(* PLC project Unnamed, Unknown Unnamed 1 *)
(* stored: creationDateTime 2021-12-21T18:23:51, modificationDateTime 2021-12-22T22:57:15 *)

TYPE datatype0 : ARRAY[1..10] OF BYTE;
END_TYPE

FUNCTION_BLOCK bot_detect
  VAR_INPUT
    IN : BOOL;
  END_VAR
  VAR
    BDGENR : UINT;
    M : BOOL;
    INIT : BOOL;
  END_VAR
  VAR_OUTPUT
    OUT : UDINT;
  END_VAR

            (* Initialize our random generator *)
(* This IF is called only the first time this *)
(* block executes *)
IF INIT = 0 THEN
  {time_t t;
  srand((unsigned) time(&t))}
  INIT := 1;
END_IF;

IF M = 0 and IN = 1 THEN
  (* Using pragma to write code directly in C. *)
  (* You can access your PLC program variables using *)
  (* GetFbVar(var,...) and SetFbVar(var,val,...) calls *)
  {SetFbVar(BDGENR,rand())}
  IF BDGENR > 4000 THEN
    {SetFbVar(OUT,1)}
  END_IF;
  IF BDGENR <= 4000 THEN
    {SetFbVar(OUT,0)}
  END_IF;
END_IF;
M := IN;
          
END_FUNCTION_BLOCK

FUNCTION_BLOCK bot_size_rand_generator
  VAR_INPUT
    IN : BOOL;
  END_VAR
  VAR
    BSZGENR : UINT;
    M : BOOL;
    INIT : BOOL;
  END_VAR
  VAR_OUTPUT
    OUT : UDINT;
  END_VAR

            (* Initialize our random generator *)
(* This IF is called only the first time this *)
(* block executes *)
IF INIT = 0 THEN
  {time_t t;
  srand((unsigned) time(&t))}
  INIT := 1;
END_IF;

IF M = 0 and IN = 1 THEN
  (* Using pragma to write code directly in C. *)
  (* You can access your PLC program variables using *)
  (* GetFbVar(var,...) and SetFbVar(var,val,...) calls *)
  {SetFbVar(BSZGENR,rand())}
  IF BSZGENR > 9000 THEN
    {SetFbVar(OUT,1)}
  END_IF;
  IF BSZGENR <= 9000 THEN
    {SetFbVar(OUT,0)}
  END_IF;
END_IF;
M := IN;
          
END_FUNCTION_BLOCK

FUNCTION_BLOCK bot_state_rand_generator
  VAR_INPUT
    IN : BOOL;
  END_VAR
  VAR
    BSGENR : UINT;
    M : BOOL;
    INIT : BOOL;
  END_VAR
  VAR_OUTPUT
    OUT : UDINT;
  END_VAR

            (* Initialize our random generator *)
(* This IF is called only the first time this *)
(* block executes *)
IF INIT = 0 THEN
  {time_t t;
  srand((unsigned) time(&t))}
  INIT := 1;
END_IF;

IF M = 0 and IN = 1 THEN
  (* Using pragma to write code directly in C. *)
  (* You can access your PLC program variables using *)
  (* GetFbVar(var,...) and SetFbVar(var,val,...) calls *)
  {SetFbVar(BSGENR,rand())}
  IF BSGENR > 4000 THEN
    {SetFbVar(OUT,1)}
  END_IF;
  IF BSGENR <= 4000 THEN
    {SetFbVar(OUT,0)}
  END_IF;
END_IF;
M := IN;
          
END_FUNCTION_BLOCK

PROGRAM BottleRefill
  VAR
    Start AT %IX0.0 : BOOL;
    Stop AT %IX0.1 : BOOL;
    System_On AT %QX0.0 : BOOL;
  END_VAR
  VAR
    TON0 : TON;
    Time_On1 : TIME;
    Time_On2 : TIME;
    Bot_Detect_State : BOOL;
    bot_size_rand_generator0 : bot_size_rand_generator;
    bot_state_rand_generator0 : bot_state_rand_generator;
    Bot_Size1 : BOOL;
    Bot_Size2 : BOOL;
    Bot_Size3 : BOOL;
    Bot_Size4 : BOOL;
    Bot_Size5 : BOOL;
    first_bot_state_bit : BYTE;
    second_bot_state_bit : BYTE;
    third_bot_state_bit : BYTE;
    fourth_bot_state_bit : BYTE;
    fifth_bot_state_bit : BYTE;
    first_bot_size_bit : BYTE;
    second_bot_size_bit : BYTE;
    third_bot_size_bit : BYTE;
    fourth_bot_size_bit : BYTE;
    fifth_bot_size_bit : BYTE;
    Bit_Timer_State1 : BOOL;
    Bit_Timer_State2 : BOOL;
    Bit_Timer_State3 : BOOL;
    Bit_Timer_State4 : BOOL;
    Bot_State1 : BOOL;
    Bot_State2 : BOOL;
    Bot_State3 : BOOL;
    Bot_State4 : BOOL;
    Bot_State5 : BOOL;
    SR0 : SR;
    SR1 : SR;
    bot_detect0 : bot_detect;
    SR2 : SR;
    SR3 : SR;
    SR4 : SR;
    SR5 : SR;
    SR6 : SR;
    SR7 : SR;
  END_VAR
  VAR
    Fill_Large AT %QX0.1 : BOOL;
    Fill_Small AT %QX0.2 : BOOL;
    Pass AT %QX0.3 : BOOL;
    Discard AT %QX0.4 : BOOL;
    Up AT %QX0.5 : BOOL;
    Down AT %QX0.6 : BOOL;
    Feed_Motor AT %QX0.7 : BOOL;
  END_VAR
  VAR
    TON1 : TON;
    TON2 : TON;
  END_VAR
  VAR  (* added by the conversion: wires and edge detectors of the diagram *)
    _LT161_ENO : BOOL;
    _LT161_OUT : BOOL;
    _LT64_ENO : BOOL;
    _LT64_OUT : BOOL;
    _LT105_ENO : BOOL;
    _LT105_OUT : BOOL;
    _LT108_ENO : BOOL;
    _LT108_OUT : BOOL;
    _LT112_ENO : BOOL;
    _LT112_OUT : BOOL;
    _LT114_ENO : BOOL;
    _LT114_OUT : BOOL;
    _GT145_ENO : BOOL;
    _GT145_OUT : BOOL;
  END_VAR

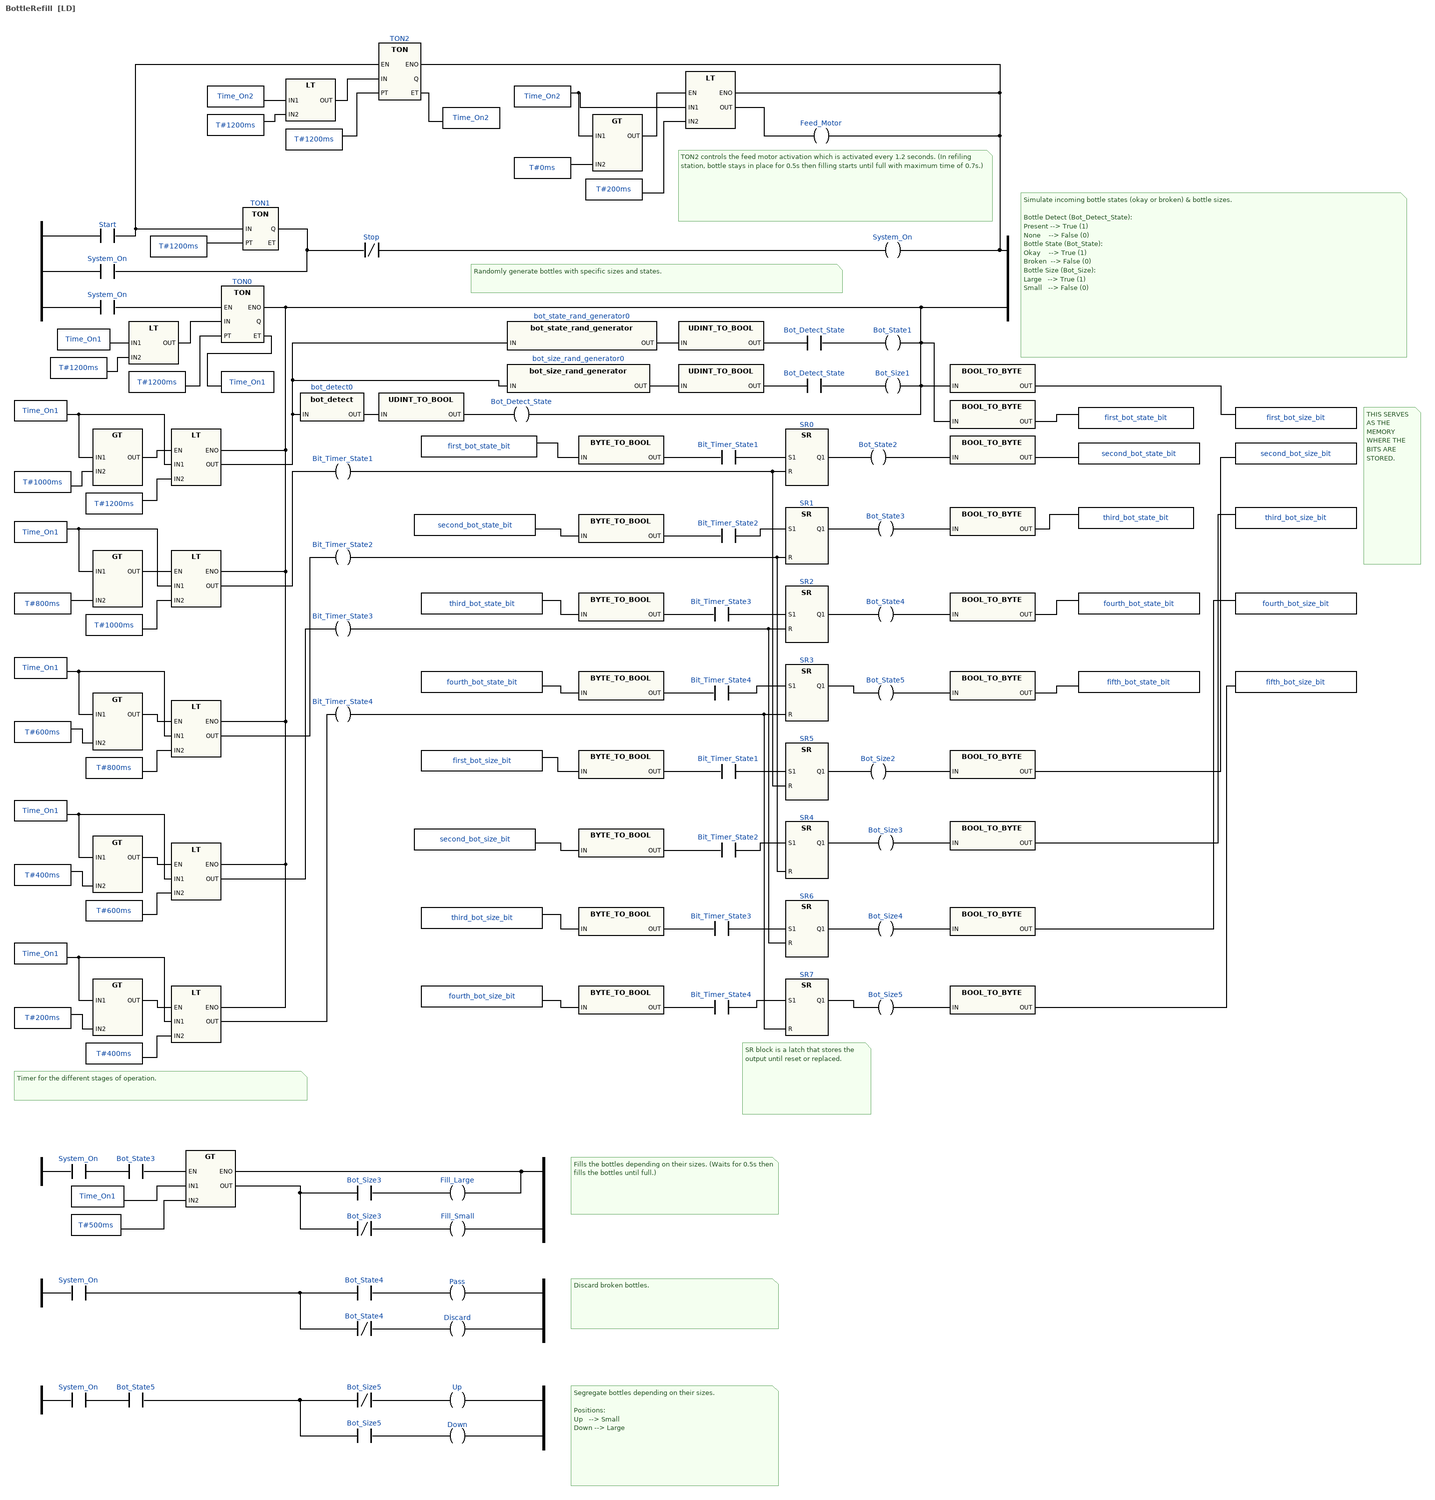
(* LD diagram, written out as Structured Text *)
TON2(EN := Start, IN := Time_On2 < T#1200ms, PT := T#1200ms);
IF TON2.ENO THEN Time_On2 := TON2.ET; END_IF;
_LT161_OUT := LT(EN := Time_On2 > T#0ms, IN1 := Time_On2, IN2 := T#200ms, ENO => _LT161_ENO);
Feed_Motor := _LT161_OUT;
(* TON2 controls the feed motor activation which is activated every 1.2 seconds. (In refiling station, bottle stays in place for 0.5s then filling starts until full with maximum time of 0.7s.) *)
(* Simulate incoming bottle states (okay or broken) & bottle sizes.

Bottle Detect (Bot_Detect_State):
     Present --> True (1)
     None    --> False (0)
Bottle State (Bot_State):
     Okay    --> True (1)
     Broken  --> False (0)
Bottle Size (Bot_Size):
     Large   --> True (1)
     Small   --> False (0) *)
TON1(IN := Start, PT := T#1200ms);
System_On := (TON1.Q OR System_On) AND NOT Stop;
(* Randomly generate bottles with specific sizes and states. *)
_LT64_OUT := LT(EN := Time_On1 > T#1000ms, IN1 := Time_On1, IN2 := T#1200ms, ENO => _LT64_ENO);
bot_state_rand_generator0(IN := _LT64_OUT);
Bot_State1 := UDINT_TO_BOOL(bot_state_rand_generator0.OUT) AND Bot_Detect_State;
TON0(EN := System_On, IN := Time_On1 < T#1200ms, PT := T#1200ms);
IF TON0.ENO THEN Time_On1 := TON0.ET; END_IF;
bot_size_rand_generator0(IN := _LT64_OUT);
Bot_Size1 := UDINT_TO_BOOL(bot_size_rand_generator0.OUT) AND Bot_Detect_State;
(* THIS SERVES AS THE MEMORY WHERE THE BITS ARE STORED. *)
bot_detect0(IN := _LT64_OUT);
Bot_Detect_State := UDINT_TO_BOOL(bot_detect0.OUT);
first_bot_state_bit := BOOL_TO_BYTE(UDINT_TO_BOOL(bot_state_rand_generator0.OUT) AND Bot_Detect_State);
first_bot_size_bit := BOOL_TO_BYTE(UDINT_TO_BOOL(bot_size_rand_generator0.OUT) AND Bot_Detect_State);
_LT105_OUT := LT(EN := Time_On1 > T#800ms, IN1 := Time_On1, IN2 := T#1000ms, ENO => _LT105_ENO);
SR0(S1 := BYTE_TO_BOOL(first_bot_state_bit) AND Bit_Timer_State1, R := _LT105_OUT);
second_bot_state_bit := BOOL_TO_BYTE(SR0.Q1);
SR5(S1 := BYTE_TO_BOOL(first_bot_size_bit) AND Bit_Timer_State1, R := _LT105_OUT);
second_bot_size_bit := BOOL_TO_BYTE(SR5.Q1);
Bot_State2 := SR0.Q1;
Bit_Timer_State1 := _LT105_OUT;
_LT108_OUT := LT(EN := Time_On1 > T#600ms, IN1 := Time_On1, IN2 := T#800ms, ENO => _LT108_ENO);
SR1(S1 := BYTE_TO_BOOL(second_bot_state_bit) AND Bit_Timer_State2, R := _LT108_OUT);
third_bot_state_bit := BOOL_TO_BYTE(SR1.Q1);
SR4(S1 := BYTE_TO_BOOL(second_bot_size_bit) AND Bit_Timer_State2, R := _LT108_OUT);
third_bot_size_bit := BOOL_TO_BYTE(SR4.Q1);
Bot_State3 := SR1.Q1;
Bit_Timer_State2 := _LT108_OUT;
_LT112_OUT := LT(EN := Time_On1 > T#400ms, IN1 := Time_On1, IN2 := T#600ms, ENO => _LT112_ENO);
SR2(S1 := BYTE_TO_BOOL(third_bot_state_bit) AND Bit_Timer_State3, R := _LT112_OUT);
fourth_bot_state_bit := BOOL_TO_BYTE(SR2.Q1);
SR6(S1 := BYTE_TO_BOOL(third_bot_size_bit) AND Bit_Timer_State3, R := _LT112_OUT);
fourth_bot_size_bit := BOOL_TO_BYTE(SR6.Q1);
Bot_State4 := SR2.Q1;
Bit_Timer_State3 := _LT112_OUT;
_LT114_OUT := LT(EN := Time_On1 > T#200ms, IN1 := Time_On1, IN2 := T#400ms, ENO => _LT114_ENO);
SR3(S1 := BYTE_TO_BOOL(fourth_bot_state_bit) AND Bit_Timer_State4, R := _LT114_OUT);
fifth_bot_state_bit := BOOL_TO_BYTE(SR3.Q1);
SR7(S1 := BYTE_TO_BOOL(fourth_bot_size_bit) AND Bit_Timer_State4, R := _LT114_OUT);
fifth_bot_size_bit := BOOL_TO_BYTE(SR7.Q1);
Bot_State5 := SR3.Q1;
Bit_Timer_State4 := _LT114_OUT;
Bot_Size2 := SR5.Q1;
Bot_Size3 := SR4.Q1;
Bot_Size4 := SR6.Q1;
Bot_Size5 := SR7.Q1;
(* SR block is a latch that stores the output until reset or replaced. *)
(* Timer for the different stages of operation. *)
(* Fills the bottles depending on their sizes. (Waits for 0.5s then fills the bottles until full.) *)
_GT145_OUT := GT(EN := System_On AND Bot_State3, IN1 := Time_On1, IN2 := T#500ms, ENO => _GT145_ENO);
Fill_Large := _GT145_OUT AND Bot_Size3;
Fill_Small := _GT145_OUT AND NOT Bot_Size3;
(* Discard broken bottles. *)
Pass := System_On AND Bot_State4;
Discard := System_On AND NOT Bot_State4;
(* Segregate bottles depending on their sizes.

Positions:
     Up   --> Small
     Down --> Large *)
Up := System_On AND Bot_State5 AND NOT Bot_Size5;
Down := System_On AND Bot_State5 AND Bot_Size5;
END_PROGRAM

CONFIGURATION Config0
  RESOURCE Res0 ON PLC
    TASK task0(INTERVAL := T#20ms, PRIORITY := 0);
    PROGRAM instance0 WITH task0 : BottleRefill;
  END_RESOURCE
END_CONFIGURATION
